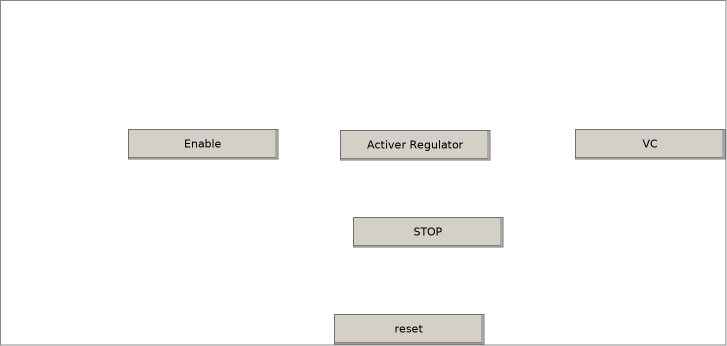
VISUALIZATION VisualizationVirtuel  // 727x346
    Button (128,129 150x30), "Enable"
        toggle PLC_PRG.enable_virtuel
    Button (340,130 150x30), "Activer Regulator"
        toggle plc_prg.activer_regulator
    Button (575,129 150x30), "VC"
        toggle plc_prg.VC_virtuel
    Button (334,314 150x30), "reset"
        toggle plc_prg.Reset
    Button (353,217 150x30), "STOP"
        toggle plc_prg.MCSTOP
END_VISUALIZATION

(* text list TextList (id | default)
   |  *)
